TYPE WrappedComponentExample_Control EXTENDS TcoCore.TcoStruct:
STRUCT

		Setpoint:INT;
		
END_STRUCT
END_TYPE

(* stored: Version 1.1.0.1
   DUT WrappedComponentExample_Control: Id {7040aa76-9333-4a97-921e-6f0133f845cb} *)
